# B&R Automation Studio project Project
Automation Studio 4.10

## Configuration BufferedFub

CPU PC_any, AutomationRuntime B4.92, Build 6.3.0, Vc V4.72.5

### Task classes (Cpu.sw)
```
Cyclic#1 (cycle 10000 us, tolerance 0 us):
  BufferFub_ <- BufferedFub.BufferFub_c-api_c-api.BufferFub_0.prg
  BufferF2_ <- BufferedFub.BufferFub2_c-api_c-api.BufferFub2_0.prg
Binaries: FWRules, udbdef, TCData, target, arconfig, User, sysconf, Role, iomap, asfw, ashwac, ashwd, components
Libraries: BufferFub, ExData, runtime, FileIO, AsIoTime, sys_lib, astime, exos, asieccon, exdeploy, astcp, BufferFub2
```

### Hardware
```
PC : PC_any v1.1.1.0 (OrderNumber=PC)
  ConfigurationID = Project_BufferedFub
  Cyclic1Duration = 10000
  Cyclic1Tolerance = 0
  Cyclic2Duration = 20000
  Cyclic2Tolerance = 0
  FileDevice1
  FileDeviceName1 = USER
  FileDevicePath1 = USER_PATH
  ActivateOpcUa = 1
  OpcUaPort = 4841
  OpcUaInformationModels_PV_Version = 1
```

### components.exoscomponent - PC/exosTechnology/components.exoscomponent
```
Element gBufferFub_0 (Type=exoscomponent)
  PackageSelection = Logical\BufferedFub\BufferFub_c-api_c-api\BufferFub.exospkg
  ErrorHandling = Component
  RestartEvent = Component
  StartupTimeout = 0
  Predefined:
    Files:
      File[0]:
        FileName = Linux\exos-comp-bufferfub_1.0.0_amd64.deb
        ChangeEvent = Reinstall
    Services:
      Service[0]:
        Type = Runtime
        Command = ./bufferfub
        WorkingDirectory = /home/user/bufferfub
      Service[1]:
        Type = Install
        Command = dpkg -i exos-comp-bufferfub_1.0.0_amd64.deb
        WorkingDirectory
      Service[2]:
        Type = Remove
        Command = dpkg --purge exos-comp-bufferfub
        WorkingDirectory
Element gBufferFub2_0 (Type=exoscomponent)
  PackageSelection = Logical\BufferedFub\BufferFub2_c-api_c-api\BufferFub2.exospkg
  ErrorHandling = Component
  RestartEvent = Component
  StartupTimeout = 0
  Predefined:
    Files:
      File[0]:
        FileName = Linux\exos-comp-bufferfub2_1.0.0_amd64.deb
        ChangeEvent = Reinstall
    Services:
      Service[0]:
        Type = Runtime
        Command = ./bufferfub2
        WorkingDirectory = /home/user/bufferfub2
      Service[1]:
        Type = Install
        Command = dpkg -i exos-comp-bufferfub2_1.0.0_amd64.deb
        WorkingDirectory
      Service[2]:
        Type = Remove
        Command = dpkg --purge exos-comp-bufferfub2
        WorkingDirectory
```

### target.exostarget - PC/exosTechnology/target.exostarget
```
Element gTarget_0 (Type=exostarget)
  General:
    ConnectionIP = 192.168.137.2
    Logging:
      LogLevel = Debug
      LogFilters:
        LogFilterUser = On
        LogFilterSystem = On
        LogFilterVerbose = On
      LogDestination = Volatile
    Deployment = On
      MaxRestarts = 10
    DataConnection = On
      ConnectionType = SharedMemory
      TimeSynchronization:
        TimeConnection:
          TimePort = 49001
        PrecisionUsec = 100
        GuardTimeSec = 4
        DeviationPerHourUsec = 100000
      DataConnectionLogging:
        LogConnection:
          LogPort = 49002
          LogShmPath = exos_log
        LogCycleTimeMsec = 100
  Components:
    ComponentsGeneral:
      ComponentsHeartbeatMsec = 500
      ComponentsTimeoutSec = 2
      ComponentsTaskClass = 2
      ComponentsCycleTimeMsec = 100
    Component[0]:
      ComponentConfigurationLink = gBufferFub_0
      DataModels:
        Instance[0]:
          InstanceName = BufferFub_0
          InstanceConnection:
            InstancePort = 49003
            InstanceShmPath = BufferFub_0
    Component[1]:
      ComponentConfigurationLink = gBufferFub2_0
      DataModels:
        Instance[0]:
          InstanceName = BufferFub2_0
          InstanceConnection:
            InstancePort = 49004
            InstanceShmPath = BufferFub2_0
  ComponentDataConnection:
    Version = 2.1.0-1
    ErrorHandling = Target
    RestartEvent = Target
    StartupTimeout = 5
    Predefined:
      Files:
        File[0]:
          FileName = ufw-exos-data
          ChangeEvent = Ignore
        File[1]:
          FileName = exos-data-ufw-profile.sh
          ChangeEvent = Ignore
        File[2]:
          FileName = exos-data-ports-allow.sh
          ChangeEvent = Restart
        File[3]:
          FileName = exos-data.conf
          ChangeEvent = Restart
        File[4]:
          FileName = exos-data_2.1.0-1_amd64.deb
          ChangeEvent = Reinstall
        File[5]:
          FileName = exos-data-eth_2.1.0-1_amd64.deb
          ChangeEvent = Reinstall
        File[6]:
          FileName = exos-data-remove.sh
          ChangeEvent = Ignore
        File[7]:
          FileName = run_server.sh
          ChangeEvent = Ignore
        File[8]:
          FileName = setup_build_environment.sh
          ChangeEvent = Ignore
        File[9]:
          FileName = libzmq5_4.2.1-4+deb9u2_amd64.deb
          ChangeEvent = Reinstall
        File[10]:
          FileName = libpgm-5.2-0_5.2.122~dfsg-2_amd64.deb
          ChangeEvent = Reinstall
        File[11]:
          FileName = libsodium18_1.0.11-2_amd64.deb
          ChangeEvent = Reinstall
      Services:
        Service[0]:
          Type = Install
          Command = dpkg -i *.deb
          WorkingDirectory
        Service[1]:
          Type = Remove
          Command = dpkg --purge exos-data
          WorkingDirectory
        Service[2]:
          Type = Remove
          Command = dpkg --purge exos-data-eth
          WorkingDirectory
        Service[3]:
          Type = Remove
          Command = sh exos-data-remove.sh
          WorkingDirectory
        Service[4]:
          Type = Startup
          Command = cp exos-data.conf /etc/exos-data.conf
          WorkingDirectory
        Service[5]:
          Type = Startup
          Command = sh exos-data-ufw-profile.sh
          WorkingDirectory
        Service[6]:
          Type = Startup
          Command = sh exos-data-ports-allow.sh
          WorkingDirectory
        Service[7]:
          Type = Runtime
          Command = /usr/bin/exos_mr
          WorkingDirectory
  Simulation:
    SimConnectionIP = 127.0.0.1
    SimDeployment = On
    SimDataConnection = On
      SimConnectionType = TCPIP
      SimTimeSynchronization:
        SimPrecisionUsec = 1000000
        SimGuardTimeSec = 30
    SimComponentsGeneral:
      SimComponentsHeartbeatMsec = 1000
      SimComponentsTimeoutSec = 75
```

## Logical view

- BufferFub.exospkg - exOS package description (not shown)

### Program Logical/BufferedFub/BufferFub_c-api_c-api/BufferFub_0 (IEC) - BufferFub application

#### BufferFub.var - BufferFub variable declaration
```iecst
VAR
    BufferFubInit_0 : BufferFubInit;
    BufferFubCyclic_0 : BufferFubCyclic;
    BufferFubExit_0 : BufferFubExit;
    BufferFubBufferUpdate_0 : BufferFubBufferUpdate;
    BufferFub_0 : BufferFub;
    ExComponentInfo_0 : ExComponentInfo;
    ExDatamodelInfo_0 : ExDatamodelInfo;
END_VAR
```

#### BufferFub.st - BufferFub application
```iecst
PROGRAM _INIT

    BufferFubInit_0();

END_PROGRAM

PROGRAM _CYCLIC

    //Auto connect:
    //BufferFubCyclic_0.Enable := ExComponentInfo_0.Operational; // Component has been deployed and started up successfully

    BufferFubCyclic_0(Handle := BufferFubInit_0.Handle, pBufferFub := ADR(BufferFub_0));

    BufferFubBufferUpdate_0.BufferHandle := BufferFubInit_0.bufferedSampleBufferHandle;
    UpdateBufferSampleSingle;
    //UpdateBufferSampleAll;

    ExComponentInfo_0(ExTargetLink := ADR(gTarget_0), ExComponentLink := ADR(gBufferFub_0), Enable := TRUE);

    ExDatamodelInfo_0(ExTargetLink := ADR(gTarget_0), Enable := TRUE, InstanceName := 'BufferFub_0');

END_PROGRAM

PROGRAM _EXIT

    BufferFubExit_0(Handle := BufferFubInit_0.Handle);

END_PROGRAM
```

#### UpdateBufferActions.st - BufferFub buffer actions
```iecst
(*Read a single change on BufferFubBufferUpdate_0.BufferHandle per scan*)
ACTION UpdateBufferSampleSingle:
    BufferFubBufferUpdate_0(UpdateDataset := TRUE);

    IF BufferFubBufferUpdate_0.DatasetUpdated THEN

        (* Your code here *)

    END_IF
END_ACTION

(*Read all changes on BufferFubBufferUpdate_0.BufferHandle within a single scan*)
ACTION UpdateBufferSampleAll:

    BufferFubBufferUpdate_0(UpdateDataset := FALSE); // update PendingUpdates without requesting UpdateDataset

    WHILE BufferFubBufferUpdate_0.PendingUpdates > 0 DO

        BufferFubBufferUpdate_0(UpdateDataset := TRUE);

        (* Your code here *)

    END_WHILE
END_ACTION
```

### Library Logical/BufferedFub/BufferFub_c-api_c-api/BufferFub (ANSIC) - BufferFub exOS library
Depends on: ExData

#### BufferFub.fun - BufferFub function blocks
```iecst
FUNCTION_BLOCK BufferFubInit
	VAR_OUTPUT
		Handle : UDINT;
		bufferedSampleBufferHandle : UDINT; (*Initialized BufferHandle for bufferedSample. Bufferhandle is linked to data in Cyclic*)
	END_VAR
	VAR
		_state : USINT;
	END_VAR
END_FUNCTION_BLOCK

FUNCTION_BLOCK BufferFubCyclic
	VAR_INPUT
		Enable : BOOL;
		Handle : UDINT;
		Start : BOOL;
		pBufferFub : REFERENCE TO BufferFub;
	END_VAR
	VAR_OUTPUT
		Active : BOOL;
		Error : BOOL;
		Disconnected : BOOL;
		Connected : BOOL;
		Operational : BOOL;
		Aborted : BOOL;
	END_VAR
	VAR
		_state : USINT;
	END_VAR
END_FUNCTION_BLOCK

FUNCTION_BLOCK BufferFubExit
	VAR_INPUT
		Handle : UDINT;
	END_VAR
	VAR
		_state : USINT;
	END_VAR
END_FUNCTION_BLOCK

FUNCTION_BLOCK BufferFubBufferUpdate (*Must be called in same TC as Cyclic. This function block finalizes in one scan and can be used for several different buffers*)
	VAR_INPUT
		BufferHandle : UDINT; (*Set this to the correct bufferhandle (from Init function block) before calling action UpdateBufferSampleSingle or UpdateBufferSampleAll*)
		UpdateDataset : BOOL; (*Set to TRUE to update dataset, PendingUpdates and OverflowErrors. Set to FALSE to only update PendingUpdates and OverflowErrors for BufferHandle without updating dataset*)
	END_VAR
	VAR_OUTPUT
		Error : BOOL; (*Set in case BufferHandle is invalid*)
		DatasetUpdated : BOOL; (*Set if dataset was updated successfully. Only when UpdateDataset is set to TRUE and there is something in the buffer*)
		PendingUpdates : UDINT; (*Number of datasets waiting in the buffer*)
		OverflowErrors : UDINT; (*Number of overflow errors which occurs when the buffer is full and new data arrives from GPOS*)
	END_VAR
END_FUNCTION_BLOCK
```

#### bufferfub.c - BufferFub library source
```c
#include <BufferFub.h>

#define EXOS_ASSERT_LOG &handle->logger
#define EXOS_ASSERT_CALLBACK inst->_state = 255;
#include "exos_log.h"
#include "exos_bufferfub.h"
#include <string.h>

#define SUCCESS(_format_, ...) exos_log_success(&handle->logger, EXOS_LOG_TYPE_USER, _format_, ##__VA_ARGS__);
#define INFO(_format_, ...) exos_log_info(&handle->logger, EXOS_LOG_TYPE_USER, _format_, ##__VA_ARGS__);
#define VERBOSE(_format_, ...) exos_log_debug(&handle->logger, EXOS_LOG_TYPE_USER + EXOS_LOG_TYPE_VERBOSE, _format_, ##__VA_ARGS__);
#define ERROR(_format_, ...) exos_log_error(&handle->logger, _format_, ##__VA_ARGS__);

typedef struct
{
    void *self;
    void* pData;
    size_t dataSize;
    void* databuffer;
    size_t bufferSize;
    size_t head;
    size_t tail;
    size_t overflowErrors;
} BufferFubBufferHandle_t;

typedef struct
{
    void *self;
    exos_log_handle_t logger;
    BufferFub data;

    exos_datamodel_handle_t bufferfub;

    exos_dataset_handle_t bufferedsample;
    BufferFubBufferHandle_t bufferedsample_buffer;
    exos_dataset_handle_t setup_dataset;
    exos_dataset_handle_t cmdsendburst;
} BufferFubHandle_t;

static int BufferFubBufferPush(BufferFubBufferHandle_t* bufferHandle, void* data)
{
    if (NULL == bufferHandle)
    {
        return -1;
    }
    if ((void *)bufferHandle != bufferHandle->self)
    {
        return -1;
    }
    if (((bufferHandle->head + 1) % bufferHandle->bufferSize) == bufferHandle->tail)
    {
        return -1;
    }

    memcpy(bufferHandle->databuffer + (bufferHandle->head * bufferHandle->dataSize), data, bufferHandle->dataSize);
    bufferHandle->head = (bufferHandle->head + 1) % bufferHandle->bufferSize;

    return 0;
}

static void datasetEvent(exos_dataset_handle_t *dataset, EXOS_DATASET_EVENT_TYPE event_type, void *info)
{
    struct BufferFubCyclic *inst = (struct BufferFubCyclic *)dataset->datamodel->user_context;
    BufferFubHandle_t *handle = (BufferFubHandle_t *)inst->Handle;

    switch (event_type)
    {
    case EXOS_DATASET_EVENT_UPDATED:
        VERBOSE("dataset %s updated! latency (us):%i", dataset->name, (exos_datamodel_get_nettime(dataset->datamodel) - dataset->nettime));
        //handle each subscription dataset separately
        if(0 == strcmp(dataset->name, "bufferedSample"))
        {
            //inst->pBufferFub->bufferedSample = *(UDINT *)dataset->data;

            if(BufferFubBufferPush(&handle->bufferedsample_buffer, dataset->data))
            {
                handle->bufferedsample_buffer.overflowErrors++;
                ERROR("Buffer overflow in bufferedSample update");
            }
        }
        break;

    case EXOS_DATASET_EVENT_PUBLISHED:
        VERBOSE("dataset %s published to local server for distribution! send buffer free:%i", dataset->name, dataset->send_buffer.free);
        //handle each published dataset separately
        if(0 == strcmp(dataset->name, "setup"))
        {
            // BufferFubSetup_typ *setup_dataset = (BufferFubSetup_typ *)dataset->data;
        }
        else if(0 == strcmp(dataset->name, "cmdSendBurst"))
        {
            // BOOL *cmdsendburst = (BOOL *)dataset->data;
        }
        break;

    case EXOS_DATASET_EVENT_DELIVERED:
        VERBOSE("dataset %s delivered to remote server for distribution! send buffer free:%i", dataset->name, dataset->send_buffer.free);
        //handle each published dataset separately
        if(0 == strcmp(dataset->name, "setup"))
        {
            // BufferFubSetup_typ *setup_dataset = (BufferFubSetup_typ *)dataset->data;
        }
        else if(0 == strcmp(dataset->name, "cmdSendBurst"))
        {
            // BOOL *cmdsendburst = (BOOL *)dataset->data;
        }
        break;

    case EXOS_DATASET_EVENT_CONNECTION_CHANGED:
        INFO("dataset %s changed state to %s", dataset->name, exos_get_state_string(dataset->connection_state));

        switch (dataset->connection_state)
        {
        case EXOS_STATE_DISCONNECTED:
            break;
        case EXOS_STATE_CONNECTED:
            //call the dataset changed event to update the dataset when connected
            //datasetEvent(dataset,EXOS_DATASET_UPDATED,info);
            break;
        case EXOS_STATE_OPERATIONAL:
            break;
        case EXOS_STATE_ABORTED:
            ERROR("dataset %s error %d (%s) occured", dataset->name, dataset->error, exos_get_error_string(dataset->error));
            break;
        }
        break;
    }

}

static void datamodelEvent(exos_datamodel_handle_t *datamodel, const EXOS_DATAMODEL_EVENT_TYPE event_type, void *info)
{
    struct BufferFubCyclic *inst = (struct BufferFubCyclic *)datamodel->user_context;
    BufferFubHandle_t *handle = (BufferFubHandle_t *)inst->Handle;

    switch (event_type)
    {
    case EXOS_DATAMODEL_EVENT_CONNECTION_CHANGED:
        INFO("application changed state to %s", exos_get_state_string(datamodel->connection_state));

        inst->Disconnected = 0;
        inst->Connected = 0;
        inst->Operational = 0;
        inst->Aborted = 0;

        switch (datamodel->connection_state)
        {
        case EXOS_STATE_DISCONNECTED:
            inst->Disconnected = 1;
            inst->_state = 255;
            break;
        case EXOS_STATE_CONNECTED:
            inst->Connected = 1;
            break;
        case EXOS_STATE_OPERATIONAL:
            SUCCESS("BufferFub operational!");
            inst->Operational = 1;
            break;
        case EXOS_STATE_ABORTED:
            ERROR("application error %d (%s) occured", datamodel->error, exos_get_error_string(datamodel->error));
            inst->_state = 255;
            inst->Aborted = 1;
            break;
        }
        break;
    case EXOS_DATAMODEL_EVENT_SYNC_STATE_CHANGED:
        break;

    default:
        break;

    }

}

_BUR_PUBLIC void BufferFubInit(struct BufferFubInit *inst)
{
    BufferFubHandle_t *handle;
    TMP_alloc(sizeof(BufferFubHandle_t), (void **)&handle);
    if (NULL == handle)
    {
        inst->Handle = 0;
        return;
    }

    memset(&handle->data, 0, sizeof(handle->data));
    handle->self = handle;

    // buffered alloc
    handle->bufferedsample_buffer.pData = 0; // set in BufferFubCyclic
    handle->bufferedsample_buffer.dataSize = sizeof(handle->data.bufferedSample);
    handle->bufferedsample_buffer.bufferSize = 20; // Note that empty is head==tail, thus only bufferSize-1 entries may be used.
    TMP_alloc(handle->bufferedsample_buffer.dataSize * handle->bufferedsample_buffer.bufferSize, (void **)&handle->bufferedsample_buffer.databuffer);
    if (NULL == handle->bufferedsample_buffer.databuffer)
    {
        inst->bufferedSampleBufferHandle = 0;
        TMP_free(sizeof(BufferFubHandle_t), (void *)handle);
        inst->Handle = 0;
        return;
    }

    handle->bufferedsample_buffer.head = 0;
    handle->bufferedsample_buffer.tail = 0;
    handle->bufferedsample_buffer.overflowErrors = 0;
    memset(handle->bufferedsample_buffer.databuffer, 0, handle->bufferedsample_buffer.dataSize * handle->bufferedsample_buffer.bufferSize);
    inst->bufferedSampleBufferHandle = &handle->bufferedsample_buffer;
    handle->bufferedsample_buffer.self = &handle->bufferedsample_buffer;

    exos_log_init(&handle->logger, "gBufferFub_0");

    exos_datamodel_handle_t *bufferfub = &handle->bufferfub;
    exos_dataset_handle_t *bufferedsample = &handle->bufferedsample;
    exos_dataset_handle_t *setup_dataset = &handle->setup_dataset;
    exos_dataset_handle_t *cmdsendburst = &handle->cmdsendburst;
    EXOS_ASSERT_OK(exos_datamodel_init(bufferfub, "BufferFub_0", "gBufferFub_0"));

    EXOS_ASSERT_OK(exos_dataset_init(bufferedsample, bufferfub, "bufferedSample", &handle->data.bufferedSample, sizeof(handle->data.bufferedSample)));
    EXOS_ASSERT_OK(exos_dataset_init(setup_dataset, bufferfub, "setup", &handle->data.setup, sizeof(handle->data.setup)));
    EXOS_ASSERT_OK(exos_dataset_init(cmdsendburst, bufferfub, "cmdSendBurst", &handle->data.cmdSendBurst, sizeof(handle->data.cmdSendBurst)));

    inst->Handle = (UDINT)handle;
}

_BUR_PUBLIC void BufferFubBufferUpdate(struct BufferFubBufferUpdate* inst)
{
    inst->DatasetUpdated = false;
    inst->Error = false;
    inst->OverflowErrors = 0;
    inst->PendingUpdates = 0;

    BufferFubBufferHandle_t *bufferHandle =  (BufferFubBufferHandle_t *)inst->BufferHandle;
    if (NULL == bufferHandle)
    {
        inst->Error = true;
        return;
    }
    if ((void *)bufferHandle != bufferHandle->self)
    {
        inst->Error = true;
        return;
    }

    inst->Error = false;
    inst->OverflowErrors = bufferHandle->overflowErrors;

    if(inst->UpdateDataset)
    {
        if (bufferHandle->tail == bufferHandle->head) // empty
        {
            inst->DatasetUpdated = false;
        }
        else
        {
            if(NULL != bufferHandle->pData)
            {
                memcpy(bufferHandle->pData, bufferHandle->databuffer + (bufferHandle->tail * bufferHandle->dataSize), bufferHandle->dataSize);
                //void* handle = bufferHandle->data[bufferHandle->tail];
                //should we set 0? bufferHandle->data[bufferHandle->tail] = NULL;
                bufferHandle->tail = (bufferHandle->tail + 1) % bufferHandle->bufferSize;
                inst->DatasetUpdated = true;
            }
            else
            {
                inst->Error = true;
                inst->DatasetUpdated = false;
            }
        }
    }
    else
    {
        inst->DatasetUpdated = false;
    }

    if (bufferHandle->tail > bufferHandle->head)
        inst->PendingUpdates = bufferHandle->bufferSize - (bufferHandle->tail - bufferHandle->head);
    else
        inst->PendingUpdates = bufferHandle->head - bufferHandle->tail;
}

_BUR_PUBLIC void BufferFubCyclic(struct BufferFubCyclic *inst)
{
    BufferFubHandle_t *handle = (BufferFubHandle_t *)inst->Handle;

    inst->Error = false;
    if (NULL == handle || NULL == inst->pBufferFub)
    {
        inst->Error = true;
        return;
    }
    if ((void *)handle != handle->self)
    {
        inst->Error = true;
        return;
    }

    // setup buffer address for xUpdate FUB:
    handle->bufferedsample_buffer.pData = &inst->pBufferFub->bufferedSample;

    BufferFub *data = &handle->data;
    exos_datamodel_handle_t *bufferfub = &handle->bufferfub;
    //the user context of the datamodel points to the BufferFubCyclic instance
    bufferfub->user_context = inst; //set it cyclically in case the program using the FUB is retransferred
    bufferfub->user_tag = 0; //user defined
    //handle online download of the library
    if(NULL != bufferfub->datamodel_event_callback && bufferfub->datamodel_event_callback != datamodelEvent)
    {
        bufferfub->datamodel_event_callback = datamodelEvent;
        exos_log_delete(&handle->logger);
        exos_log_init(&handle->logger, "gBufferFub_0");
    }

    exos_dataset_handle_t *bufferedsample = &handle->bufferedsample;
    bufferedsample->user_context = NULL; //user defined
    bufferedsample->user_tag = 0; //user defined
    //handle online download of the library
    if(NULL != bufferedsample->dataset_event_callback && bufferedsample->dataset_event_callback != datasetEvent)
    {
        bufferedsample->dataset_event_callback = datasetEvent;
    }

    exos_dataset_handle_t *setup_dataset = &handle->setup_dataset;
    setup_dataset->user_context = NULL; //user defined
    setup_dataset->user_tag = 0; //user defined
    //handle online download of the library
    if(NULL != setup_dataset->dataset_event_callback && setup_dataset->dataset_event_callback != datasetEvent)
    {
        setup_dataset->dataset_event_callback = datasetEvent;
    }

    exos_dataset_handle_t *cmdsendburst = &handle->cmdsendburst;
    cmdsendburst->user_context = NULL; //user defined
    cmdsendburst->user_tag = 0; //user defined
    //handle online download of the library
    if(NULL != cmdsendburst->dataset_event_callback && cmdsendburst->dataset_event_callback != datasetEvent)
    {
        cmdsendburst->dataset_event_callback = datasetEvent;
    }

    //unregister on disable
    if (inst->_state && !inst->Enable)
    {
        inst->_state = 255;
    }

    switch (inst->_state)
    {
    case 0:
        inst->Disconnected = 1;
        inst->Connected = 0;
        inst->Operational = 0;
        inst->Aborted = 0;

        if (inst->Enable)
        {
            inst->_state = 10;
        }
        break;

    case 10:
        inst->_state = 100;

        SUCCESS("starting BufferFub application..");

        //connect the datamodel, then the datasets
        EXOS_ASSERT_OK(exos_datamodel_connect_bufferfub(bufferfub, datamodelEvent));
        EXOS_ASSERT_OK(exos_dataset_connect(bufferedsample, EXOS_DATASET_SUBSCRIBE, datasetEvent));
        EXOS_ASSERT_OK(exos_dataset_connect(setup_dataset, EXOS_DATASET_PUBLISH, datasetEvent));
        EXOS_ASSERT_OK(exos_dataset_connect(cmdsendburst, EXOS_DATASET_PUBLISH, datasetEvent));

        inst->Active = true;
        break;

    case 100:
    case 101:
        if (inst->Start)
        {
            if (inst->_state == 100)
            {
                EXOS_ASSERT_OK(exos_datamodel_set_operational(bufferfub));
                inst->_state = 101;
            }
        }
        else
        {
            inst->_state = 100;
        }

        EXOS_ASSERT_OK(exos_datamodel_process(bufferfub));
        //put your cyclic code here!

        //publish the setup_dataset dataset as soon as there are changes
        if (0 != memcmp(&inst->pBufferFub->setup, &data->setup, sizeof(data->setup)))
        {
            memcpy(&data->setup, &inst->pBufferFub->setup, sizeof(data->setup));
            exos_dataset_publish(setup_dataset);
        }
        //publish the cmdsendburst dataset as soon as there are changes
        if (inst->pBufferFub->cmdSendBurst != data->cmdSendBurst)
        {
            data->cmdSendBurst = inst->pBufferFub->cmdSendBurst;
            exos_dataset_publish(cmdsendburst);
        }

        break;

    case 255:
        //disconnect the datamodel
        EXOS_ASSERT_OK(exos_datamodel_disconnect(bufferfub));

        inst->Active = false;
        inst->_state = 254;
        //no break

    case 254:
        if (!inst->Enable)
            inst->_state = 0;
        break;
    }

    exos_log_process(&handle->logger);

}

_BUR_PUBLIC void BufferFubExit(struct BufferFubExit *inst)
{
    BufferFubHandle_t *handle = (BufferFubHandle_t *)inst->Handle;

    if (NULL == handle)
    {
        ERROR("BufferFubExit: NULL handle, cannot delete resources");
        return;
    }
    if ((void *)handle != handle->self)
    {
        ERROR("BufferFubExit: invalid handle, cannot delete resources");
        return;
    }

    exos_datamodel_handle_t *bufferfub = &handle->bufferfub;

    EXOS_ASSERT_OK(exos_datamodel_delete(bufferfub));

    //delete buffer:
    BufferFubBufferHandle_t *bufferHandle =  (BufferFubBufferHandle_t *)&handle->bufferedsample_buffer;
    if (NULL == bufferHandle)
    {
        ERROR("BufferFubExit: NULL bufferhandle, cannot delete resources");
        return;
    }
    if ((void *)bufferHandle != bufferHandle->self)
    {
        ERROR("BufferFubExit: invalid bufferhandle, cannot delete resources");
        return;
    }

    //finish with deleting the log
    exos_log_delete(&handle->logger);
    //free the allocated handle
    TMP_free(sizeof(BufferFubHandle_t), (void *)handle);
}
```

### Package Logical/BufferedFub/BufferFub_c-api_c-api/Linux - BufferFub Linux resources

### bufferfub.c
```c
#include <unistd.h>
#include <string.h>
#include "termination.h"

#define EXOS_ASSERT_LOG &logger
#include "exos_log.h"
#include "exos_bufferfub.h"

#define SUCCESS(_format_, ...) exos_log_success(&logger, EXOS_LOG_TYPE_USER, _format_, ##__VA_ARGS__);
#define INFO(_format_, ...) exos_log_info(&logger, EXOS_LOG_TYPE_USER, _format_, ##__VA_ARGS__);
#define VERBOSE(_format_, ...) exos_log_debug(&logger, EXOS_LOG_TYPE_USER + EXOS_LOG_TYPE_VERBOSE, _format_, ##__VA_ARGS__);
#define ERROR(_format_, ...) exos_log_error(&logger, _format_, ##__VA_ARGS__);

exos_log_handle_t logger;

typedef struct {
    BufferFub *data;

    exos_datamodel_handle_t* bufferfub;

    exos_dataset_handle_t* bufferedsample;
    exos_dataset_handle_t* setup_dataset;
    exos_dataset_handle_t* cmdsendburst;
} application_info_t;

static void datasetEvent(exos_dataset_handle_t *dataset, EXOS_DATASET_EVENT_TYPE event_type, void *info)
{
    switch (event_type)
    {
    case EXOS_DATASET_EVENT_UPDATED:
        VERBOSE("dataset %s updated! latency (us):%i", dataset->name, (exos_datamodel_get_nettime(dataset->datamodel) - dataset->nettime));
        //handle each subscription dataset separately
        if(0 == strcmp(dataset->name,"setup"))
        {
            BufferFubSetup_typ *setup_dataset = (BufferFubSetup_typ *)dataset->data;
        }
        else if(0 == strcmp(dataset->name,"cmdSendBurst"))
        {
            bool *cmdsendburst = (bool *)dataset->data;

            if (*cmdsendburst){

                application_info_t *application = (application_info_t *)dataset->user_context;
                if (NULL != application)
                {
                    VERBOSE("Send burst, sampleCount=%u, sampleDelay=%u  ", application->data->setup.sampleCount, application->data->setup.sampleDelay);

                    for (size_t i = 0; i < application->data->setup.sampleCount; i++)
                    {
                        application->data->bufferedSample = i + 1;
                        exos_dataset_publish(application->bufferedsample);

                        usleep(application->data->setup.sampleDelay);
                    }
                }
            }
        }
        break;

    case EXOS_DATASET_EVENT_PUBLISHED:
        VERBOSE("dataset %s published to local server for distribution! send buffer free:%i", dataset->name, dataset->send_buffer.free);
        //handle each published dataset separately
        if(0 == strcmp(dataset->name, "bufferedSample"))
        {
            uint32_t *bufferedsample = (uint32_t *)dataset->data;
        }
        break;

    case EXOS_DATASET_EVENT_DELIVERED:
        VERBOSE("dataset %s delivered to remote server for distribution! send buffer free:%i", dataset->name, dataset->send_buffer.free);
        //handle each published dataset separately
        if(0 == strcmp(dataset->name, "bufferedSample"))
        {
            uint32_t *bufferedsample = (uint32_t *)dataset->data;
        }
        break;

    case EXOS_DATASET_EVENT_CONNECTION_CHANGED:
        INFO("dataset %s changed state to %s", dataset->name, exos_get_state_string(dataset->connection_state));

        switch (dataset->connection_state)
        {
        case EXOS_STATE_DISCONNECTED:
            break;
        case EXOS_STATE_CONNECTED:
            //call the dataset changed event to update the dataset when connected
            //datasetEvent(dataset,EXOS_DATASET_UPDATED,info);
            break;
        case EXOS_STATE_OPERATIONAL:
            break;
        case EXOS_STATE_ABORTED:
            ERROR("dataset %s error %d (%s) occured", dataset->name, dataset->error, exos_get_error_string(dataset->error));
            break;
        }
        break;
    }

}

static void datamodelEvent(exos_datamodel_handle_t *datamodel, const EXOS_DATAMODEL_EVENT_TYPE event_type, void *info)
{
    switch (event_type)
    {
    case EXOS_DATAMODEL_EVENT_CONNECTION_CHANGED:
        INFO("application changed state to %s", exos_get_state_string(datamodel->connection_state));

        switch (datamodel->connection_state)
        {
        case EXOS_STATE_DISCONNECTED:
            break;
        case EXOS_STATE_CONNECTED:
            break;
        case EXOS_STATE_OPERATIONAL:
            SUCCESS("BufferFub operational!");
            break;
        case EXOS_STATE_ABORTED:
            ERROR("application error %d (%s) occured", datamodel->error, exos_get_error_string(datamodel->error));
            break;
        }
        break;
    case EXOS_DATAMODEL_EVENT_SYNC_STATE_CHANGED:
        break;

    default:
        break;

    }

}

int main()
{
    BufferFub data;

    exos_datamodel_handle_t bufferfub;

    exos_dataset_handle_t bufferedsample;
    exos_dataset_handle_t setup_dataset;
    exos_dataset_handle_t cmdsendburst;

    application_info_t myapplication = {&data, &bufferfub, &bufferedsample, &setup_dataset, &cmdsendburst};

    exos_log_init(&logger, "gBufferFub_0");

    SUCCESS("starting BufferFub application..");

    EXOS_ASSERT_OK(exos_datamodel_init(&bufferfub, "BufferFub_0", "gBufferFub_0"));

    //set the user_context to access custom data in the callbacks
    bufferfub.user_context = NULL; //user defined
    bufferfub.user_tag = 0; //user defined

    EXOS_ASSERT_OK(exos_dataset_init(&bufferedsample, &bufferfub, "bufferedSample", &data.bufferedSample, sizeof(data.bufferedSample)));
    bufferedsample.user_context = NULL; //user defined
    bufferedsample.user_tag = 0; //user defined

    EXOS_ASSERT_OK(exos_dataset_init(&setup_dataset, &bufferfub, "setup", &data.setup, sizeof(data.setup)));
    setup_dataset.user_context = NULL; //user defined
    setup_dataset.user_tag = 0; //user defined

    EXOS_ASSERT_OK(exos_dataset_init(&cmdsendburst, &bufferfub, "cmdSendBurst", &data.cmdSendBurst, sizeof(data.cmdSendBurst)));
    cmdsendburst.user_context = &myapplication; //user defined
    cmdsendburst.user_tag = 0; //user defined

    //connect the datamodel
    EXOS_ASSERT_OK(exos_datamodel_connect_bufferfub(&bufferfub, datamodelEvent));

    //connect datasets
    EXOS_ASSERT_OK(exos_dataset_connect(&bufferedsample, EXOS_DATASET_PUBLISH, datasetEvent));
    EXOS_ASSERT_OK(exos_dataset_connect(&setup_dataset, EXOS_DATASET_SUBSCRIBE, datasetEvent));
    EXOS_ASSERT_OK(exos_dataset_connect(&cmdsendburst, EXOS_DATASET_SUBSCRIBE, datasetEvent));

    catch_termination();
    while (true)
    {
        EXOS_ASSERT_OK(exos_datamodel_process(&bufferfub));
        exos_log_process(&logger);

        //put your cyclic code here!

        if (is_terminated())
        {
            SUCCESS("BufferFub application terminated, closing..");
            break;
        }
    }

    EXOS_ASSERT_OK(exos_datamodel_delete(&bufferfub));

    //finish with deleting the log
    exos_log_delete(&logger);
    return 0;
}
```

- BufferFub2.exospkg - exOS package description (not shown)

### Program Logical/BufferedFub/BufferFub2_c-api_c-api/BufferFub2_0 (IEC) - BufferFub2 application

#### BufferFub2.var - BufferFub2 variable declaration
```iecst
VAR
    BufferFub2Init_0 : BufferFub2Init;
    BufferFub2Cyclic_0 : BufferFub2Cyclic;
    BufferFub2Exit_0 : BufferFub2Exit;
    BufferFub2BufferUpdate_0 : BufferFub2BufferUpdate;
    BufferFub2_0 : BufferFub2;
    ExComponentInfo_0 : ExComponentInfo;
    ExDatamodelInfo_0 : ExDatamodelInfo;
END_VAR
```

#### BufferFub2.st - BufferFub2 application
```iecst
PROGRAM _INIT

    BufferFub2Init_0();

END_PROGRAM

PROGRAM _CYCLIC

    //Auto connect:
    //BufferFub2Cyclic_0.Enable := ExComponentInfo_0.Operational; // Component has been deployed and started up successfully

    BufferFub2Cyclic_0(Handle := BufferFub2Init_0.Handle, pBufferFub2 := ADR(BufferFub2_0));

    BufferFub2BufferUpdate_0.BufferHandle := BufferFub2Init_0.bufferedSampleBufferHandle;
    UpdateBufferSampleSingle;
    //UpdateBufferSampleAll;

    ExComponentInfo_0(ExTargetLink := ADR(gTarget_0), ExComponentLink := ADR(gBufferFub2_0), Enable := TRUE);

    ExDatamodelInfo_0(ExTargetLink := ADR(gTarget_0), Enable := TRUE, InstanceName := 'BufferFub2_0');

END_PROGRAM

PROGRAM _EXIT

    BufferFub2Exit_0(Handle := BufferFub2Init_0.Handle);

END_PROGRAM
```

#### UpdateBufferActions.st - BufferFub2 buffer actions
```iecst
(*Read a single change on BufferFub2BufferUpdate_0.BufferHandle per scan*)
ACTION UpdateBufferSampleSingle:
    BufferFub2BufferUpdate_0(UpdateDataset := TRUE);

    IF BufferFub2BufferUpdate_0.DatasetUpdated THEN

        (* Your code here *)

    END_IF
END_ACTION

(*Read all changes on BufferFub2BufferUpdate_0.BufferHandle within a single scan*)
ACTION UpdateBufferSampleAll:

    BufferFub2BufferUpdate_0(UpdateDataset := FALSE); // update PendingUpdates without requesting UpdateDataset

    WHILE BufferFub2BufferUpdate_0.PendingUpdates > 0 DO

        BufferFub2BufferUpdate_0(UpdateDataset := TRUE);

        (* Your code here *)

    END_WHILE
END_ACTION
```

### Library Logical/BufferedFub/BufferFub2_c-api_c-api/BufferFub2 (ANSIC) - BufferFub2 exOS library
Depends on: ExData

#### BufferFub2.typ - BufferFub2 datamodel declaration
```iecst
TYPE
	BufferFub2Setup_typ : 	STRUCT
		sampleCount : UDINT; (*number of samples sent each time cmdSendBurst is set*)
		sampleDelay : UDINT; (*ms between samples*)
	END_STRUCT;
	BufferFub2SubStruct_typ : 	STRUCT
		moreid : UDINT; (*id number*)
		moredata : REAL; (*some data*)
	END_STRUCT;
	BufferFub2Sample_typ : 	STRUCT
		id : UDINT; (*id number*)
		data : REAL; (*some data*)
		subStruct : BufferFub2SubStruct_typ; (*a sub structure*)
	END_STRUCT;
	BufferFub2 : 	STRUCT
		bufferedSample : BufferFub2Sample_typ; (*SUB BUFFERED*)
		setup : BufferFub2Setup_typ; (*PUB*)
		cmdSendBurst : BOOL; (*PUB*)
	END_STRUCT;
END_TYPE
```

#### BufferFub2.fun - BufferFub2 function blocks
```iecst
FUNCTION_BLOCK BufferFub2Init
	VAR_OUTPUT
		Handle : UDINT;
		bufferedSampleBufferHandle : UDINT; (*Initialized BufferHandle for bufferedSample. Bufferhandle is linked to data in Cyclic*)
	END_VAR
	VAR
		_state : USINT;
	END_VAR
END_FUNCTION_BLOCK

FUNCTION_BLOCK BufferFub2Cyclic
	VAR_INPUT
		Enable : BOOL;
		Handle : UDINT;
		Start : BOOL;
		pBufferFub2 : REFERENCE TO BufferFub2;
	END_VAR
	VAR_OUTPUT
		Active : BOOL;
		Error : BOOL;
		Disconnected : BOOL;
		Connected : BOOL;
		Operational : BOOL;
		Aborted : BOOL;
	END_VAR
	VAR
		_state : USINT;
	END_VAR
END_FUNCTION_BLOCK

FUNCTION_BLOCK BufferFub2Exit
	VAR_INPUT
		Handle : UDINT;
	END_VAR
	VAR
		_state : USINT;
	END_VAR
END_FUNCTION_BLOCK

FUNCTION_BLOCK BufferFub2BufferUpdate (*Must be called in same TC as Cyclic. This function block finalizes in one scan and can be used for several different buffers*)
	VAR_INPUT
		BufferHandle : UDINT; (*Set this to the correct bufferhandle (from Init function block) before calling action UpdateBufferSampleSingle or UpdateBufferSampleAll*)
		UpdateDataset : BOOL; (*Set to TRUE to update dataset, PendingUpdates and OverflowErrors. Set to FALSE to only update PendingUpdates and OverflowErrors for BufferHandle without updating dataset*)
	END_VAR
	VAR_OUTPUT
		Error : BOOL; (*Set in case BufferHandle is invalid*)
		DatasetUpdated : BOOL; (*Set if dataset was updated successfully. Only when UpdateDataset is set to TRUE and there is something in the buffer*)
		PendingUpdates : UDINT; (*Number of datasets waiting in the buffer*)
		OverflowErrors : UDINT; (*Number of overflow errors which occurs when the buffer is full and new data arrives from GPOS*)
	END_VAR
END_FUNCTION_BLOCK
```

#### bufferfub2.c - BufferFub2 library source
```c
#include <BufferFub2.h>

#define EXOS_ASSERT_LOG &handle->logger
#define EXOS_ASSERT_CALLBACK inst->_state = 255;
#include "exos_log.h"
#include "exos_bufferfub2.h"
#include <string.h>

#define SUCCESS(_format_, ...) exos_log_success(&handle->logger, EXOS_LOG_TYPE_USER, _format_, ##__VA_ARGS__);
#define INFO(_format_, ...) exos_log_info(&handle->logger, EXOS_LOG_TYPE_USER, _format_, ##__VA_ARGS__);
#define VERBOSE(_format_, ...) exos_log_debug(&handle->logger, EXOS_LOG_TYPE_USER + EXOS_LOG_TYPE_VERBOSE, _format_, ##__VA_ARGS__);
#define ERROR(_format_, ...) exos_log_error(&handle->logger, _format_, ##__VA_ARGS__);

typedef struct
{
    void *self;
    void* pData;
    size_t dataSize;
    void* databuffer;
    size_t bufferSize;
    size_t head;
    size_t tail;
    size_t overflowErrors;
} BufferFub2BufferHandle_t;

typedef struct
{
    void *self;
    exos_log_handle_t logger;
    BufferFub2 data;

    exos_datamodel_handle_t bufferfub2;

    exos_dataset_handle_t bufferedsample;
    BufferFub2BufferHandle_t bufferedsample_buffer;
    exos_dataset_handle_t setup_dataset;
    exos_dataset_handle_t cmdsendburst;
} BufferFub2Handle_t;

static int BufferFub2BufferPush(BufferFub2BufferHandle_t* bufferHandle, void* data)
{
    if (NULL == bufferHandle)
    {
        return -1;
    }
    if ((void *)bufferHandle != bufferHandle->self)
    {
        return -1;
    }
    if (((bufferHandle->head + 1) % bufferHandle->bufferSize) == bufferHandle->tail)
    {
        return -1;
    }

    memcpy(bufferHandle->databuffer + (bufferHandle->head * bufferHandle->dataSize), data, bufferHandle->dataSize);
    bufferHandle->head = (bufferHandle->head + 1) % bufferHandle->bufferSize;

    return 0;
}

static void datasetEvent(exos_dataset_handle_t *dataset, EXOS_DATASET_EVENT_TYPE event_type, void *info)
{
    struct BufferFub2Cyclic *inst = (struct BufferFub2Cyclic *)dataset->datamodel->user_context;
    BufferFub2Handle_t *handle = (BufferFub2Handle_t *)inst->Handle;

    switch (event_type)
    {
    case EXOS_DATASET_EVENT_UPDATED:
        VERBOSE("dataset %s updated! latency (us):%i", dataset->name, (exos_datamodel_get_nettime(dataset->datamodel) - dataset->nettime));
        //handle each subscription dataset separately
        if(0 == strcmp(dataset->name, "bufferedSample"))
        {
            if(BufferFub2BufferPush(&handle->bufferedsample_buffer, dataset->data))
            {
                handle->bufferedsample_buffer.overflowErrors++;
                ERROR("Buffer overflow in bufferedSample update");
            }
        }
        break;

    case EXOS_DATASET_EVENT_PUBLISHED:
        VERBOSE("dataset %s published to local server for distribution! send buffer free:%i", dataset->name, dataset->send_buffer.free);
        //handle each published dataset separately
        if(0 == strcmp(dataset->name, "setup"))
        {
            // BufferFub2Setup_typ *setup_dataset = (BufferFub2Setup_typ *)dataset->data;
        }
        else if(0 == strcmp(dataset->name, "cmdSendBurst"))
        {
            // BOOL *cmdsendburst = (BOOL *)dataset->data;
        }
        break;

    case EXOS_DATASET_EVENT_DELIVERED:
        VERBOSE("dataset %s delivered to remote server for distribution! send buffer free:%i", dataset->name, dataset->send_buffer.free);
        //handle each published dataset separately
        if(0 == strcmp(dataset->name, "setup"))
        {
            // BufferFub2Setup_typ *setup_dataset = (BufferFub2Setup_typ *)dataset->data;
        }
        else if(0 == strcmp(dataset->name, "cmdSendBurst"))
        {
            // BOOL *cmdsendburst = (BOOL *)dataset->data;
        }
        break;

    case EXOS_DATASET_EVENT_CONNECTION_CHANGED:
        INFO("dataset %s changed state to %s", dataset->name, exos_get_state_string(dataset->connection_state));

        switch (dataset->connection_state)
        {
        case EXOS_STATE_DISCONNECTED:
            break;
        case EXOS_STATE_CONNECTED:
            //call the dataset changed event to update the dataset when connected
            //datasetEvent(dataset,EXOS_DATASET_UPDATED,info);
            break;
        case EXOS_STATE_OPERATIONAL:
            break;
        case EXOS_STATE_ABORTED:
            ERROR("dataset %s error %d (%s) occured", dataset->name, dataset->error, exos_get_error_string(dataset->error));
            break;
        }
        break;
    }

}

static void datamodelEvent(exos_datamodel_handle_t *datamodel, const EXOS_DATAMODEL_EVENT_TYPE event_type, void *info)
{
    struct BufferFub2Cyclic *inst = (struct BufferFub2Cyclic *)datamodel->user_context;
    BufferFub2Handle_t *handle = (BufferFub2Handle_t *)inst->Handle;

    switch (event_type)
    {
    case EXOS_DATAMODEL_EVENT_CONNECTION_CHANGED:
        INFO("application changed state to %s", exos_get_state_string(datamodel->connection_state));

        inst->Disconnected = 0;
        inst->Connected = 0;
        inst->Operational = 0;
        inst->Aborted = 0;

        switch (datamodel->connection_state)
        {
        case EXOS_STATE_DISCONNECTED:
            inst->Disconnected = 1;
            inst->_state = 255;
            break;
        case EXOS_STATE_CONNECTED:
            inst->Connected = 1;
            break;
        case EXOS_STATE_OPERATIONAL:
            SUCCESS("BufferFub2 operational!");
            inst->Operational = 1;
            break;
        case EXOS_STATE_ABORTED:
            ERROR("application error %d (%s) occured", datamodel->error, exos_get_error_string(datamodel->error));
            inst->_state = 255;
            inst->Aborted = 1;
            break;
        }
        break;
    case EXOS_DATAMODEL_EVENT_SYNC_STATE_CHANGED:
        break;

    default:
        break;

    }

}

_BUR_PUBLIC void BufferFub2Init(struct BufferFub2Init *inst)
{
    BufferFub2Handle_t *handle;
    TMP_alloc(sizeof(BufferFub2Handle_t), (void **)&handle);
    if (NULL == handle)
    {
        inst->Handle = 0;
        return;
    }

    memset(&handle->data, 0, sizeof(handle->data));
    handle->self = handle;

    // Allocation and initialization of buffer(s)
    handle->bufferedsample_buffer.pData = 0; // set in BufferFub2Cyclic
    handle->bufferedsample_buffer.dataSize = sizeof(handle->data.bufferedSample);
    handle->bufferedsample_buffer.bufferSize = 20; // Note that empty is head==tail, thus only bufferSize-1 entries may be used.
    TMP_alloc(handle->bufferedsample_buffer.dataSize * handle->bufferedsample_buffer.bufferSize, (void **)&handle->bufferedsample_buffer.databuffer);
    if (NULL == handle->bufferedsample_buffer.databuffer)
    {
        inst->bufferedSampleBufferHandle = 0;
        TMP_free(sizeof(BufferFub2Handle_t), (void *)handle);
        inst->Handle = 0;
        return;
    }

    handle->bufferedsample_buffer.head = 0;
    handle->bufferedsample_buffer.tail = 0;
    handle->bufferedsample_buffer.overflowErrors = 0;
    memset(handle->bufferedsample_buffer.databuffer, 0, handle->bufferedsample_buffer.dataSize * handle->bufferedsample_buffer.bufferSize);
    inst->bufferedSampleBufferHandle = (UDINT)&handle->bufferedsample_buffer;
    handle->bufferedsample_buffer.self = &handle->bufferedsample_buffer;

    exos_log_init(&handle->logger, "gBufferFub2_0");

    exos_datamodel_handle_t *bufferfub2 = &handle->bufferfub2;
    exos_dataset_handle_t *bufferedsample = &handle->bufferedsample;
    exos_dataset_handle_t *setup_dataset = &handle->setup_dataset;
    exos_dataset_handle_t *cmdsendburst = &handle->cmdsendburst;
    EXOS_ASSERT_OK(exos_datamodel_init(bufferfub2, "BufferFub2_0", "gBufferFub2_0"));

    EXOS_ASSERT_OK(exos_dataset_init(bufferedsample, bufferfub2, "bufferedSample", &handle->data.bufferedSample, sizeof(handle->data.bufferedSample)));
    EXOS_ASSERT_OK(exos_dataset_init(setup_dataset, bufferfub2, "setup", &handle->data.setup, sizeof(handle->data.setup)));
    EXOS_ASSERT_OK(exos_dataset_init(cmdsendburst, bufferfub2, "cmdSendBurst", &handle->data.cmdSendBurst, sizeof(handle->data.cmdSendBurst)));

    inst->Handle = (UDINT)handle;
}

_BUR_PUBLIC void BufferFub2BufferUpdate(struct BufferFub2BufferUpdate* inst)
{
    inst->DatasetUpdated = false;
    inst->Error = false;
    inst->OverflowErrors = 0;
    inst->PendingUpdates = 0;

    BufferFub2BufferHandle_t *bufferHandle =  (BufferFub2BufferHandle_t *)inst->BufferHandle;
    if (NULL == bufferHandle)
    {
        inst->Error = true;
        return;
    }
    if ((void *)bufferHandle != bufferHandle->self)
    {
        inst->Error = true;
        return;
    }

    inst->Error = false;
    inst->OverflowErrors = bufferHandle->overflowErrors;

    if(inst->UpdateDataset)
    {
        if (bufferHandle->tail == bufferHandle->head) // empty
        {
            inst->DatasetUpdated = false;
        }
        else
        {
            if(NULL != bufferHandle->pData)
            {
                memcpy(bufferHandle->pData, bufferHandle->databuffer + (bufferHandle->tail * bufferHandle->dataSize), bufferHandle->dataSize);
                //void* handle = bufferHandle->data[bufferHandle->tail];
                //should we set 0? bufferHandle->data[bufferHandle->tail] = NULL;
                bufferHandle->tail = (bufferHandle->tail + 1) % bufferHandle->bufferSize;
                inst->DatasetUpdated = true;
            }
            else
            {
                inst->Error = true;
                inst->DatasetUpdated = false;
            }
        }
    }
    else
    {
        inst->DatasetUpdated = false;
    }

    if (bufferHandle->tail > bufferHandle->head)
        inst->PendingUpdates = bufferHandle->bufferSize - (bufferHandle->tail - bufferHandle->head);
    else
        inst->PendingUpdates = bufferHandle->head - bufferHandle->tail;
}

_BUR_PUBLIC void BufferFub2Cyclic(struct BufferFub2Cyclic *inst)
{
    BufferFub2Handle_t *handle = (BufferFub2Handle_t *)inst->Handle;

    inst->Error = false;
    if (NULL == handle || NULL == inst->pBufferFub2)
    {
        inst->Error = true;
        return;
    }
    if ((void *)handle != handle->self)
    {
        inst->Error = true;
        return;
    }

    // setup buffer address(es) for BufferFub2Update:
    handle->bufferedsample_buffer.pData = &inst->pBufferFub2->bufferedSample;

    BufferFub2 *data = &handle->data;
    exos_datamodel_handle_t *bufferfub2 = &handle->bufferfub2;
    //the user context of the datamodel points to the BufferFub2Cyclic instance
    bufferfub2->user_context = inst; //set it cyclically in case the program using the FUB is retransferred
    bufferfub2->user_tag = 0; //user defined
    //handle online download of the library
    if(NULL != bufferfub2->datamodel_event_callback && bufferfub2->datamodel_event_callback != datamodelEvent)
    {
        bufferfub2->datamodel_event_callback = datamodelEvent;
        exos_log_delete(&handle->logger);
        exos_log_init(&handle->logger, "gBufferFub2_0");
    }

    exos_dataset_handle_t *bufferedsample = &handle->bufferedsample;
    bufferedsample->user_context = NULL; //user defined
    bufferedsample->user_tag = 0; //user defined
    //handle online download of the library
    if(NULL != bufferedsample->dataset_event_callback && bufferedsample->dataset_event_callback != datasetEvent)
    {
        bufferedsample->dataset_event_callback = datasetEvent;
    }

    exos_dataset_handle_t *setup_dataset = &handle->setup_dataset;
    setup_dataset->user_context = NULL; //user defined
    setup_dataset->user_tag = 0; //user defined
    //handle online download of the library
    if(NULL != setup_dataset->dataset_event_callback && setup_dataset->dataset_event_callback != datasetEvent)
    {
        setup_dataset->dataset_event_callback = datasetEvent;
    }

    exos_dataset_handle_t *cmdsendburst = &handle->cmdsendburst;
    cmdsendburst->user_context = NULL; //user defined
    cmdsendburst->user_tag = 0; //user defined
    //handle online download of the library
    if(NULL != cmdsendburst->dataset_event_callback && cmdsendburst->dataset_event_callback != datasetEvent)
    {
        cmdsendburst->dataset_event_callback = datasetEvent;
    }

    //unregister on disable
    if (inst->_state && !inst->Enable)
    {
        inst->_state = 255;
    }

    switch (inst->_state)
    {
    case 0:
        inst->Disconnected = 1;
        inst->Connected = 0;
        inst->Operational = 0;
        inst->Aborted = 0;

        if (inst->Enable)
        {
            inst->_state = 10;
        }
        break;

    case 10:
        inst->_state = 100;

        SUCCESS("starting BufferFub2 application..");

        //connect the datamodel, then the datasets
        EXOS_ASSERT_OK(exos_datamodel_connect_bufferfub2(bufferfub2, datamodelEvent));
        EXOS_ASSERT_OK(exos_dataset_connect(bufferedsample, EXOS_DATASET_SUBSCRIBE, datasetEvent));
        EXOS_ASSERT_OK(exos_dataset_connect(setup_dataset, EXOS_DATASET_PUBLISH, datasetEvent));
        EXOS_ASSERT_OK(exos_dataset_connect(cmdsendburst, EXOS_DATASET_PUBLISH, datasetEvent));

        inst->Active = true;
        break;

    case 100:
    case 101:
        if (inst->Start)
        {
            if (inst->_state == 100)
            {
                EXOS_ASSERT_OK(exos_datamodel_set_operational(bufferfub2));
                inst->_state = 101;
            }
        }
        else
        {
            inst->_state = 100;
        }

        EXOS_ASSERT_OK(exos_datamodel_process(bufferfub2));
        //put your cyclic code here!

        //publish the setup_dataset dataset as soon as there are changes
        if (0 != memcmp(&inst->pBufferFub2->setup, &data->setup, sizeof(data->setup)))
        {
            memcpy(&data->setup, &inst->pBufferFub2->setup, sizeof(data->setup));
            exos_dataset_publish(setup_dataset);
        }
        //publish the cmdsendburst dataset as soon as there are changes
        if (inst->pBufferFub2->cmdSendBurst != data->cmdSendBurst)
        {
            data->cmdSendBurst = inst->pBufferFub2->cmdSendBurst;
            exos_dataset_publish(cmdsendburst);
        }

        break;

    case 255:
        //disconnect the datamodel
        EXOS_ASSERT_OK(exos_datamodel_disconnect(bufferfub2));

        inst->Active = false;
        inst->_state = 254;
        //no break

    case 254:
        if (!inst->Enable)
            inst->_state = 0;
        break;
    }

    exos_log_process(&handle->logger);

}

_BUR_PUBLIC void BufferFub2Exit(struct BufferFub2Exit *inst)
{
    BufferFub2Handle_t *handle = (BufferFub2Handle_t *)inst->Handle;

    if (NULL == handle)
    {
        ERROR("BufferFub2Exit: NULL handle, cannot delete resources");
        return;
    }
    if ((void *)handle != handle->self)
    {
        ERROR("BufferFub2Exit: invalid handle, cannot delete resources");
        return;
    }

    exos_datamodel_handle_t *bufferfub2 = &handle->bufferfub2;

    EXOS_ASSERT_OK(exos_datamodel_delete(bufferfub2));

    //delete buffer(s):
    BufferFub2BufferHandle_t *bufferHandle =  (BufferFub2BufferHandle_t *)&handle->bufferedsample_buffer;
    if (NULL == bufferHandle)
    {
        ERROR("BufferFub2Exit: NULL bufferhandle, cannot delete resources");
        return;
    }
    if ((void *)bufferHandle != bufferHandle->self)
    {
        ERROR("BufferFub2Exit: invalid bufferhandle, cannot delete resources");
        return;
    }

    //finish with deleting the log
    exos_log_delete(&handle->logger);
    //free the allocated handle
    TMP_free(sizeof(BufferFub2Handle_t), (void *)handle);
}
```

### Package Logical/BufferedFub/BufferFub2_c-api_c-api/Linux - BufferFub2 Linux resources

### exos_bufferfub2.h - Generated datamodel header for BufferFub2
```c
/*Automatically generated header file from BufferFub2.typ*/

#ifndef _EXOS_COMP_BUFFERFUB2_H_
#define _EXOS_COMP_BUFFERFUB2_H_

#include "exos_api.h"

#if defined(_SG4)
#include <BufferFub2.h>
#else
#include <stddef.h>
#include <stdint.h>
#include <stdbool.h>

typedef struct BufferFub2Setup_typ
{
    uint32_t sampleCount; //number of samples sent each time cmdSendBurst is set
    uint32_t sampleDelay; //ms between samples

} BufferFub2Setup_typ;

typedef struct BufferFub2SubStruct_typ
{
    uint32_t moreid; //id number
    float moredata; //some data

} BufferFub2SubStruct_typ;

typedef struct BufferFub2Sample_typ
{
    uint32_t id; //id number
    float data; //some data
    struct BufferFub2SubStruct_typ subStruct; //a sub structure

} BufferFub2Sample_typ;

typedef struct BufferFub2
{
    struct BufferFub2Sample_typ bufferedSample; //SUB BUFFERED
    struct BufferFub2Setup_typ setup; //PUB
    bool cmdSendBurst; //PUB

} BufferFub2;

#endif // _SG4

EXOS_ERROR_CODE exos_datamodel_connect_bufferfub2(exos_datamodel_handle_t *datamodel, exos_datamodel_event_cb datamodel_event_callback);

#endif // _EXOS_COMP_BUFFERFUB2_H_
```

### exos_bufferfub2.c - Generated datamodel source for BufferFub2
```c
/*Automatically generated c file from BufferFub2.typ*/

#include "exos_bufferfub2.h"

const char config_bufferfub2[] = "{\"name\":\"struct\",\"attributes\":{\"name\":\"<NAME>\",\"dataType\":\"BufferFub2\",\"info\":\"<infoId0>\"},\"children\":[{\"name\":\"struct\",\"attributes\":{\"name\":\"bufferedSample\",\"dataType\":\"BufferFub2Sample_typ\",\"comment\":\"SUB\",\"info\":\"<infoId1>\"},\"children\":[{\"name\":\"variable\",\"attributes\":{\"name\":\"id\",\"dataType\":\"UDINT\",\"info\":\"<infoId2>\"}},{\"name\":\"variable\",\"attributes\":{\"name\":\"data\",\"dataType\":\"REAL\",\"info\":\"<infoId3>\"}},{\"name\":\"struct\",\"attributes\":{\"name\":\"subStruct\",\"dataType\":\"BufferFub2SubStruct_typ\",\"info\":\"<infoId4>\"},\"children\":[{\"name\":\"variable\",\"attributes\":{\"name\":\"moreid\",\"dataType\":\"UDINT\",\"info\":\"<infoId5>\"}},{\"name\":\"variable\",\"attributes\":{\"name\":\"moredata\",\"dataType\":\"REAL\",\"info\":\"<infoId6>\"}}]}]},{\"name\":\"struct\",\"attributes\":{\"name\":\"setup\",\"dataType\":\"BufferFub2Setup_typ\",\"comment\":\"PUB\",\"info\":\"<infoId7>\"},\"children\":[{\"name\":\"variable\",\"attributes\":{\"name\":\"sampleCount\",\"dataType\":\"UDINT\",\"info\":\"<infoId8>\"}},{\"name\":\"variable\",\"attributes\":{\"name\":\"sampleDelay\",\"dataType\":\"UDINT\",\"info\":\"<infoId9>\"}}]},{\"name\":\"variable\",\"attributes\":{\"name\":\"cmdSendBurst\",\"dataType\":\"BOOL\",\"comment\":\"PUB\",\"info\":\"<infoId10>\"}}]}";

/*Connect the BufferFub2 datamodel to the server*/
EXOS_ERROR_CODE exos_datamodel_connect_bufferfub2(exos_datamodel_handle_t *datamodel, exos_datamodel_event_cb datamodel_event_callback)
{
    BufferFub2 data;
    exos_dataset_info_t datasets[] = {
        {EXOS_DATASET_BROWSE_NAME_INIT,{}},
        {EXOS_DATASET_BROWSE_NAME(bufferedSample),{}},
        {EXOS_DATASET_BROWSE_NAME(bufferedSample.id),{}},
        {EXOS_DATASET_BROWSE_NAME(bufferedSample.data),{}},
        {EXOS_DATASET_BROWSE_NAME(bufferedSample.subStruct),{}},
        {EXOS_DATASET_BROWSE_NAME(bufferedSample.subStruct.moreid),{}},
        {EXOS_DATASET_BROWSE_NAME(bufferedSample.subStruct.moredata),{}},
        {EXOS_DATASET_BROWSE_NAME(setup),{}},
        {EXOS_DATASET_BROWSE_NAME(setup.sampleCount),{}},
        {EXOS_DATASET_BROWSE_NAME(setup.sampleDelay),{}},
        {EXOS_DATASET_BROWSE_NAME(cmdSendBurst),{}}
    };

    exos_datamodel_calc_dataset_info(datasets, sizeof(datasets));

    return exos_datamodel_connect(datamodel, config_bufferfub2, datasets, sizeof(datasets), datamodel_event_callback);
}
```

### bufferfub2.c - Linux application
```c
#include <unistd.h>
#include <string.h>
#include "termination.h"

#define EXOS_ASSERT_LOG &logger
#include "exos_log.h"
#include "exos_bufferfub2.h"

#define SUCCESS(_format_, ...) exos_log_success(&logger, EXOS_LOG_TYPE_USER, _format_, ##__VA_ARGS__);
#define INFO(_format_, ...) exos_log_info(&logger, EXOS_LOG_TYPE_USER, _format_, ##__VA_ARGS__);
#define VERBOSE(_format_, ...) exos_log_debug(&logger, EXOS_LOG_TYPE_USER + EXOS_LOG_TYPE_VERBOSE, _format_, ##__VA_ARGS__);
#define ERROR(_format_, ...) exos_log_error(&logger, _format_, ##__VA_ARGS__);

exos_log_handle_t logger;

static void datasetEvent(exos_dataset_handle_t *dataset, EXOS_DATASET_EVENT_TYPE event_type, void *info)
{
    switch (event_type)
    {
    case EXOS_DATASET_EVENT_UPDATED:
        VERBOSE("dataset %s updated! latency (us):%i", dataset->name, (exos_datamodel_get_nettime(dataset->datamodel) - dataset->nettime));
        //handle each subscription dataset separately
        if(0 == strcmp(dataset->name,"setup"))
        {
            BufferFub2Setup_typ *setup_dataset = (BufferFub2Setup_typ *)dataset->data;
        }
        else if(0 == strcmp(dataset->name,"cmdSendBurst"))
        {
            bool *cmdsendburst = (bool *)dataset->data;
        }
        break;

    case EXOS_DATASET_EVENT_PUBLISHED:
        VERBOSE("dataset %s published to local server for distribution! send buffer free:%i", dataset->name, dataset->send_buffer.free);
        //handle each published dataset separately
        if(0 == strcmp(dataset->name, "bufferedSample"))
        {
            BufferFub2Sample_typ *bufferedsample = (BufferFub2Sample_typ *)dataset->data;
        }
        break;

    case EXOS_DATASET_EVENT_DELIVERED:
        VERBOSE("dataset %s delivered to remote server for distribution! send buffer free:%i", dataset->name, dataset->send_buffer.free);
        //handle each published dataset separately
        if(0 == strcmp(dataset->name, "bufferedSample"))
        {
            BufferFub2Sample_typ *bufferedsample = (BufferFub2Sample_typ *)dataset->data;
        }
        break;

    case EXOS_DATASET_EVENT_CONNECTION_CHANGED:
        INFO("dataset %s changed state to %s", dataset->name, exos_get_state_string(dataset->connection_state));

        switch (dataset->connection_state)
        {
        case EXOS_STATE_DISCONNECTED:
            break;
        case EXOS_STATE_CONNECTED:
            //call the dataset changed event to update the dataset when connected
            //datasetEvent(dataset,EXOS_DATASET_UPDATED,info);
            break;
        case EXOS_STATE_OPERATIONAL:
            break;
        case EXOS_STATE_ABORTED:
            ERROR("dataset %s error %d (%s) occured", dataset->name, dataset->error, exos_get_error_string(dataset->error));
            break;
        }
        break;
    }

}

static void datamodelEvent(exos_datamodel_handle_t *datamodel, const EXOS_DATAMODEL_EVENT_TYPE event_type, void *info)
{
    switch (event_type)
    {
    case EXOS_DATAMODEL_EVENT_CONNECTION_CHANGED:
        INFO("application changed state to %s", exos_get_state_string(datamodel->connection_state));

        switch (datamodel->connection_state)
        {
        case EXOS_STATE_DISCONNECTED:
            break;
        case EXOS_STATE_CONNECTED:
            break;
        case EXOS_STATE_OPERATIONAL:
            SUCCESS("BufferFub2 operational!");
            break;
        case EXOS_STATE_ABORTED:
            ERROR("application error %d (%s) occured", datamodel->error, exos_get_error_string(datamodel->error));
            break;
        }
        break;
    case EXOS_DATAMODEL_EVENT_SYNC_STATE_CHANGED:
        break;

    default:
        break;

    }

}

int main()
{
    BufferFub2 data;

    exos_datamodel_handle_t bufferfub2;

    exos_dataset_handle_t bufferedsample;
    exos_dataset_handle_t setup_dataset;
    exos_dataset_handle_t cmdsendburst;

    exos_log_init(&logger, "gBufferFub2_0");

    SUCCESS("starting BufferFub2 application..");

    EXOS_ASSERT_OK(exos_datamodel_init(&bufferfub2, "BufferFub2_0", "gBufferFub2_0"));

    //set the user_context to access custom data in the callbacks
    bufferfub2.user_context = NULL; //user defined
    bufferfub2.user_tag = 0; //user defined

    EXOS_ASSERT_OK(exos_dataset_init(&bufferedsample, &bufferfub2, "bufferedSample", &data.bufferedSample, sizeof(data.bufferedSample)));
    bufferedsample.user_context = NULL; //user defined
    bufferedsample.user_tag = 0; //user defined

    EXOS_ASSERT_OK(exos_dataset_init(&setup_dataset, &bufferfub2, "setup", &data.setup, sizeof(data.setup)));
    setup_dataset.user_context = NULL; //user defined
    setup_dataset.user_tag = 0; //user defined

    EXOS_ASSERT_OK(exos_dataset_init(&cmdsendburst, &bufferfub2, "cmdSendBurst", &data.cmdSendBurst, sizeof(data.cmdSendBurst)));
    cmdsendburst.user_context = NULL; //user defined
    cmdsendburst.user_tag = 0; //user defined

    //connect the datamodel
    EXOS_ASSERT_OK(exos_datamodel_connect_bufferfub2(&bufferfub2, datamodelEvent));

    //connect datasets
    EXOS_ASSERT_OK(exos_dataset_connect(&bufferedsample, EXOS_DATASET_PUBLISH, datasetEvent));
    EXOS_ASSERT_OK(exos_dataset_connect(&setup_dataset, EXOS_DATASET_SUBSCRIBE, datasetEvent));
    EXOS_ASSERT_OK(exos_dataset_connect(&cmdsendburst, EXOS_DATASET_SUBSCRIBE, datasetEvent));

    catch_termination();
    while (true)
    {
        EXOS_ASSERT_OK(exos_datamodel_process(&bufferfub2));
        exos_log_process(&logger);

        //put your cyclic code here!

        if (is_terminated())
        {
            SUCCESS("BufferFub2 application terminated, closing..");
            break;
        }
    }

    EXOS_ASSERT_OK(exos_datamodel_delete(&bufferfub2));

    //finish with deleting the log
    exos_log_delete(&logger);
    return 0;
}
```

### CMakeLists.txt - CMake build file script
```
cmake_minimum_required(VERSION 3.0)

project(bufferfub2)

set(CMAKE_BUILD_TYPE Debug)
add_executable(bufferfub2 termination.c bufferfub2.c exos_bufferfub2.c)
target_include_directories(bufferfub2 PUBLIC ..)
target_link_libraries(bufferfub2 zmq exos-api)

install(TARGETS bufferfub2 RUNTIME DESTINATION /home/user/bufferfub2)

set(CPACK_GENERATOR "DEB")
set(CPACK_PACKAGE_NAME exos-comp-bufferfub2)
set(CPACK_PACKAGE_DESCRIPTION_SUMMARY "BufferFub2 summary")
set(CPACK_PACKAGE_DESCRIPTION "Some description")
set(CPACK_PACKAGE_VENDOR "Your Company")

set(CPACK_PACKAGE_VERSION_MAJOR 1)
set(CPACK_PACKAGE_VERSION_MINOR 0)
set(CPACK_PACKAGE_VERSION_PATCH 0)
set(CPACK_PACKAGE_FILE_NAME exos-comp-bufferfub2_1.0.0_amd64)
set(CPACK_DEBIAN_PACKAGE_MAINTAINER "Your Name")

set(CPACK_DEBIAN_PACKAGE_SHLIBDEPS ON)

include(CPack)
```

- build.sh - build file shell script (not shown)

- bufferfub2 - BufferFub2 application (binary file, 33072 bytes)
### Library Logical/BufferedFub/BufferFub_c-static_c-api/BufferFub (ANSIC)
Depends on: ExData

#### exos_bufferfub.h - Generated datamodel header for BufferFub
```c
/*Automatically generated header file from BufferFub.typ*/

#ifndef _EXOS_COMP_BUFFERFUB_H_
#define _EXOS_COMP_BUFFERFUB_H_

#include "exos_api.h"

#if defined(_SG4)
#include <BufferFub.h>
#else
#include <stddef.h>
#include <stdint.h>
#include <stdbool.h>

typedef struct BufferFubSetup_typ
{
    uint32_t sampleCount; //number of samples sent each time cmdSendBurst is set
    uint32_t sampleDelay; //ms between samples

} BufferFubSetup_typ;

typedef struct BufferFub
{
    uint32_t bufferedSample; //SUB BUFFERED
    struct BufferFubSetup_typ setup; //PUB
    bool cmdSendBurst; //PUB

} BufferFub;

#endif // _SG4

EXOS_ERROR_CODE exos_datamodel_connect_bufferfub(exos_datamodel_handle_t *datamodel, exos_datamodel_event_cb datamodel_event_callback);

#endif // _EXOS_COMP_BUFFERFUB_H_
```

#### libbufferfub.h - BufferFub static library wrapper header
```c
#ifndef _LIBBUFFERFUB_H_
#define _LIBBUFFERFUB_H_

#include "exos_bufferfub.h"

typedef void (*libBufferFub_event_cb)(void);
typedef void (*libBufferFub_method_fn)(void);
typedef int32_t (*libBufferFub_get_nettime_fn)(void);
typedef void (*libBufferFub_log_fn)(char *log_entry);

typedef struct libBufferFubbufferedSample
{
    libBufferFub_event_cb on_change;
    int32_t nettime;
    uint32_t value;
} libBufferFubbufferedSample_t;

typedef struct libBufferFubsetup
{
    libBufferFub_method_fn publish;
    BufferFubSetup_typ value;
} libBufferFubsetup_t;

typedef struct libBufferFubcmdSendBurst
{
    libBufferFub_method_fn publish;
    bool value;
} libBufferFubcmdSendBurst_t;

typedef struct libBufferFub_log
{
    libBufferFub_log_fn error;
    libBufferFub_log_fn warning;
    libBufferFub_log_fn success;
    libBufferFub_log_fn info;
    libBufferFub_log_fn debug;
    libBufferFub_log_fn verbose;
} libBufferFub_log_t;

typedef struct libBufferFub
{
    libBufferFub_method_fn connect;
    libBufferFub_method_fn disconnect;
    libBufferFub_method_fn process;
    libBufferFub_method_fn set_operational;
    libBufferFub_method_fn dispose;
    libBufferFub_get_nettime_fn get_nettime;
    libBufferFub_log_t log;
    libBufferFub_event_cb on_connected;
    libBufferFub_event_cb on_disconnected;
    libBufferFub_event_cb on_operational;
    bool is_connected;
    bool is_operational;
    libBufferFubbufferedSample_t bufferedSample;
    libBufferFubsetup_t setup;
    libBufferFubcmdSendBurst_t cmdSendBurst;
} libBufferFub_t;

#ifdef __cplusplus
extern "C" {
#endif
libBufferFub_t *libBufferFub_init(void);
#ifdef __cplusplus
}
#endif
#endif // _LIBBUFFERFUB_H_
```

### Program Logical/BufferedFub/BufferFub_c-static_c-api/BufferFub_0 (IEC)

#### BufferFub.var - BufferFub variable declaration
```iecst
VAR
    BufferFub_0 : BufferFub;
    BufferFubCyclic_0 : BufferFubCyclic;
    ExComponentInfo_0 : ExComponentInfo;
    ExDatamodelInfo_0 : ExDatamodelInfo;
END_VAR
```

### Program Logical/BufferedFub/BufferFub_c-static_c-api/Linux

#### bufferfub.c
```c
#include <unistd.h>
#include <string.h>
#include "termination.h"

#define EXOS_ASSERT_LOG &logger
#include "exos_log.h"
#include "exos_bufferfub.h"

#define SUCCESS(_format_, ...) exos_log_success(&logger, EXOS_LOG_TYPE_USER, _format_, ##__VA_ARGS__);
#define INFO(_format_, ...) exos_log_info(&logger, EXOS_LOG_TYPE_USER, _format_, ##__VA_ARGS__);
#define VERBOSE(_format_, ...) exos_log_debug(&logger, EXOS_LOG_TYPE_USER + EXOS_LOG_TYPE_VERBOSE, _format_, ##__VA_ARGS__);
#define ERROR(_format_, ...) exos_log_error(&logger, _format_, ##__VA_ARGS__);

exos_log_handle_t logger;

static void datasetEvent(exos_dataset_handle_t *dataset, EXOS_DATASET_EVENT_TYPE event_type, void *info)
{
    switch (event_type)
    {
    case EXOS_DATASET_EVENT_UPDATED:
        VERBOSE("dataset %s updated! latency (us):%i", dataset->name, (exos_datamodel_get_nettime(dataset->datamodel) - dataset->nettime));
        //handle each subscription dataset separately
        if(0 == strcmp(dataset->name,"setup"))
        {
            BufferFubSetup_typ *setup_dataset = (BufferFubSetup_typ *)dataset->data;
        }
        else if(0 == strcmp(dataset->name,"cmdSendBurst"))
        {
            bool *cmdsendburst = (bool *)dataset->data;
        }
        break;

    case EXOS_DATASET_EVENT_PUBLISHED:
        VERBOSE("dataset %s published to local server for distribution! send buffer free:%i", dataset->name, dataset->send_buffer.free);
        //handle each published dataset separately
        if(0 == strcmp(dataset->name, "bufferedSample"))
        {
            uint32_t *bufferedsample = (uint32_t *)dataset->data;
        }
        break;

    case EXOS_DATASET_EVENT_DELIVERED:
        VERBOSE("dataset %s delivered to remote server for distribution! send buffer free:%i", dataset->name, dataset->send_buffer.free);
        //handle each published dataset separately
        if(0 == strcmp(dataset->name, "bufferedSample"))
        {
            uint32_t *bufferedsample = (uint32_t *)dataset->data;
        }
        break;

    case EXOS_DATASET_EVENT_CONNECTION_CHANGED:
        INFO("dataset %s changed state to %s", dataset->name, exos_get_state_string(dataset->connection_state));

        switch (dataset->connection_state)
        {
        case EXOS_STATE_DISCONNECTED:
            break;
        case EXOS_STATE_CONNECTED:
            //call the dataset changed event to update the dataset when connected
            //datasetEvent(dataset,EXOS_DATASET_UPDATED,info);
            break;
        case EXOS_STATE_OPERATIONAL:
            break;
        case EXOS_STATE_ABORTED:
            ERROR("dataset %s error %d (%s) occured", dataset->name, dataset->error, exos_get_error_string(dataset->error));
            break;
        }
        break;
    }

}

static void datamodelEvent(exos_datamodel_handle_t *datamodel, const EXOS_DATAMODEL_EVENT_TYPE event_type, void *info)
{
    switch (event_type)
    {
    case EXOS_DATAMODEL_EVENT_CONNECTION_CHANGED:
        INFO("application changed state to %s", exos_get_state_string(datamodel->connection_state));

        switch (datamodel->connection_state)
        {
        case EXOS_STATE_DISCONNECTED:
            break;
        case EXOS_STATE_CONNECTED:
            break;
        case EXOS_STATE_OPERATIONAL:
            SUCCESS("BufferFub operational!");
            break;
        case EXOS_STATE_ABORTED:
            ERROR("application error %d (%s) occured", datamodel->error, exos_get_error_string(datamodel->error));
            break;
        }
        break;
    case EXOS_DATAMODEL_EVENT_SYNC_STATE_CHANGED:
        break;

    default:
        break;

    }

}

int main()
{
    BufferFub data;

    exos_datamodel_handle_t bufferfub;

    exos_dataset_handle_t bufferedsample;
    exos_dataset_handle_t setup_dataset;
    exos_dataset_handle_t cmdsendburst;

    exos_log_init(&logger, "gBufferFub_0");

    SUCCESS("starting BufferFub application..");

    EXOS_ASSERT_OK(exos_datamodel_init(&bufferfub, "BufferFub_0", "gBufferFub_0"));

    //set the user_context to access custom data in the callbacks
    bufferfub.user_context = NULL; //user defined
    bufferfub.user_tag = 0; //user defined

    EXOS_ASSERT_OK(exos_dataset_init(&bufferedsample, &bufferfub, "bufferedSample", &data.bufferedSample, sizeof(data.bufferedSample)));
    bufferedsample.user_context = NULL; //user defined
    bufferedsample.user_tag = 0; //user defined

    EXOS_ASSERT_OK(exos_dataset_init(&setup_dataset, &bufferfub, "setup", &data.setup, sizeof(data.setup)));
    setup_dataset.user_context = NULL; //user defined
    setup_dataset.user_tag = 0; //user defined

    EXOS_ASSERT_OK(exos_dataset_init(&cmdsendburst, &bufferfub, "cmdSendBurst", &data.cmdSendBurst, sizeof(data.cmdSendBurst)));
    cmdsendburst.user_context = NULL; //user defined
    cmdsendburst.user_tag = 0; //user defined

    //connect the datamodel
    EXOS_ASSERT_OK(exos_datamodel_connect_bufferfub(&bufferfub, datamodelEvent));

    //connect datasets
    EXOS_ASSERT_OK(exos_dataset_connect(&bufferedsample, EXOS_DATASET_PUBLISH, datasetEvent));
    EXOS_ASSERT_OK(exos_dataset_connect(&setup_dataset, EXOS_DATASET_SUBSCRIBE, datasetEvent));
    EXOS_ASSERT_OK(exos_dataset_connect(&cmdsendburst, EXOS_DATASET_SUBSCRIBE, datasetEvent));

    catch_termination();
    while (true)
    {
        EXOS_ASSERT_OK(exos_datamodel_process(&bufferfub));
        exos_log_process(&logger);

        //put your cyclic code here!

        if (is_terminated())
        {
            SUCCESS("BufferFub application terminated, closing..");
            break;
        }
    }

    EXOS_ASSERT_OK(exos_datamodel_delete(&bufferfub));

    //finish with deleting the log
    exos_log_delete(&logger);
    return 0;
}
```

#### CMakeLists.txt
```
cmake_minimum_required(VERSION 3.0)

project(bufferfub)

set(CMAKE_BUILD_TYPE Debug)
add_executable(bufferfub termination.c bufferfub.c exos_bufferfub.c)
target_include_directories(bufferfub PUBLIC ..)
target_link_libraries(bufferfub zmq exos-api)

install(TARGETS bufferfub RUNTIME DESTINATION /home/user/bufferfub)

set(CPACK_GENERATOR "DEB")
set(CPACK_PACKAGE_NAME exos-comp-bufferfub)
set(CPACK_PACKAGE_DESCRIPTION_SUMMARY "BufferFub summary")
set(CPACK_PACKAGE_DESCRIPTION "Some description")
set(CPACK_PACKAGE_VENDOR "Your Company")

set(CPACK_PACKAGE_VERSION_MAJOR 1)
set(CPACK_PACKAGE_VERSION_MINOR 0)
set(CPACK_PACKAGE_VERSION_PATCH 0)
set(CPACK_PACKAGE_FILE_NAME exos-comp-bufferfub_1.0.0_amd64)
set(CPACK_DEBIAN_PACKAGE_MAINTAINER "Your Name")

set(CPACK_DEBIAN_PACKAGE_SHLIBDEPS ON)

include(CPack)
```

### Library Logical/BufferedFub/BufferFub_cpp_c-api/BufferFub (ANSIC) - BufferFub exOS library
Depends on: ExData

#### exos_bufferfub.c - Generated datamodel source for BufferFub
```c
/*Automatically generated c file from BufferFub.typ*/

#include "exos_bufferfub.h"

const char config_bufferfub[] = "{\"name\":\"struct\",\"attributes\":{\"name\":\"<NAME>\",\"dataType\":\"BufferFub\",\"info\":\"<infoId0>\"},\"children\":[{\"name\":\"variable\",\"attributes\":{\"name\":\"bufferedSample\",\"dataType\":\"UDINT\",\"comment\":\"SUB\",\"info\":\"<infoId1>\"}},{\"name\":\"struct\",\"attributes\":{\"name\":\"setup\",\"dataType\":\"BufferFubSetup_typ\",\"comment\":\"PUB\",\"info\":\"<infoId2>\"},\"children\":[{\"name\":\"variable\",\"attributes\":{\"name\":\"sampleCount\",\"dataType\":\"UDINT\",\"info\":\"<infoId3>\"}},{\"name\":\"variable\",\"attributes\":{\"name\":\"sampleDelay\",\"dataType\":\"UDINT\",\"info\":\"<infoId4>\"}}]},{\"name\":\"variable\",\"attributes\":{\"name\":\"cmdSendBurst\",\"dataType\":\"BOOL\",\"comment\":\"PUB\",\"info\":\"<infoId5>\"}}]}";

/*Connect the BufferFub datamodel to the server*/
EXOS_ERROR_CODE exos_datamodel_connect_bufferfub(exos_datamodel_handle_t *datamodel, exos_datamodel_event_cb datamodel_event_callback)
{
    BufferFub data;
    exos_dataset_info_t datasets[] = {
        {EXOS_DATASET_BROWSE_NAME_INIT,{}},
        {EXOS_DATASET_BROWSE_NAME(bufferedSample),{}},
        {EXOS_DATASET_BROWSE_NAME(setup),{}},
        {EXOS_DATASET_BROWSE_NAME(setup.sampleCount),{}},
        {EXOS_DATASET_BROWSE_NAME(setup.sampleDelay),{}},
        {EXOS_DATASET_BROWSE_NAME(cmdSendBurst),{}}
    };

    exos_datamodel_calc_dataset_info(datasets, sizeof(datasets));

    return exos_datamodel_connect(datamodel, config_bufferfub, datasets, sizeof(datasets), datamodel_event_callback);
}
```

#### BufferFubDataset.hpp - BufferFub dataset class
```cpp
#if __GNUC__ == 4
#error ########## GCC 4.1.2 used but C++ Template Requires GCC 6.3 - Change the complier in the build options ##########
#endif
#ifndef _BUFFERFUBDATASET_H_
#define _BUFFERFUBDATASET_H_

#include <string>
#include <iostream>
#include <string.h>
#include <functional>

extern "C" {
    #include "exos_bufferfub.h"
}

#include "BufferFubLogger.hpp"
#define exos_assert_ok(_plog_,_exp_)                                                                                                    \
    do                                                                                                                                  \
    {                                                                                                                                   \
        EXOS_ERROR_CODE err = _exp_;                                                                                                    \
        if (EXOS_ERROR_OK != err)                                                                                                       \
        {                                                                                                                               \
            _plog_->error << "Error in file " << __FILE__ << ":" << __LINE__ << std::endl;                                               \
            _plog_->error << #_exp_ " returned " << err << " (" << exos_get_error_string(err) << ") instead of expected 0" << std::endl; \
        }                                                                                                                               \
    } while (0)

template <typename T>
class BufferFubDataset
{
private:
    exos_dataset_handle_t dataset = {};
    BufferFubLogger* log;
    std::function<void()> _onChange = [](){};
    void datasetEvent(exos_dataset_handle_t *dataset, EXOS_DATASET_EVENT_TYPE event_type, void *info) {
        switch (event_type)
        {
            case EXOS_DATASET_EVENT_UPDATED:
                log->verbose << "dataset " << dataset->name << " updated! latency (us):" << (exos_datamodel_get_nettime(dataset->datamodel) - dataset->nettime) << std::endl;
                nettime = dataset->nettime;
                _onChange();
                break;
            case EXOS_DATASET_EVENT_PUBLISHED:
                log->verbose << "dataset " << dataset->name << "  published to local server for distribution! send buffer free:" << dataset->send_buffer.free << std::endl;
                break;
            case EXOS_DATASET_EVENT_DELIVERED:
                log->verbose << "dataset " << dataset->name << " delivered to remote server for distribution! send buffer free:" << dataset->send_buffer.free << std::endl;
                break;
            case EXOS_DATASET_EVENT_CONNECTION_CHANGED:
                log->info << "dataset " << dataset->name << " changed state to " << exos_get_state_string(dataset->connection_state) << std::endl;

                switch (dataset->connection_state)
                {
                    case EXOS_STATE_DISCONNECTED:
                        break;
                    case EXOS_STATE_CONNECTED:
                        break;
                    case EXOS_STATE_OPERATIONAL:
                        break;
                    case EXOS_STATE_ABORTED:
                        log->error << "dataset " << dataset->name << " error " << dataset->error << " (" << exos_get_error_string(dataset->error) << ") occured" << std::endl;
                        break;
                }
                break;
        }
    }
    static void _datasetEvent(exos_dataset_handle_t *dataset, EXOS_DATASET_EVENT_TYPE event_type, void *info) {
        BufferFubDataset* inst = static_cast<BufferFubDataset*>(dataset->user_context);
        inst->datasetEvent(dataset, event_type, info);
    }

public:
    BufferFubDataset() {};

    T value;
    int nettime;
    void init(exos_datamodel_handle_t *datamodel, const char *browse_name, BufferFubLogger* _log) {
        log = _log;
        exos_assert_ok(log, exos_dataset_init(&dataset, datamodel, browse_name, &value, sizeof(value)));
        dataset.user_context = this;
    };
    void connect(EXOS_DATASET_TYPE type) {
        exos_assert_ok(log, exos_dataset_connect(&dataset, type, &BufferFubDataset::_datasetEvent));
    };
    void publish() {
        exos_dataset_publish(&dataset);
    };
    void onChange(std::function<void()> f) {_onChange = std::move(f);};

    ~BufferFubDataset() {
        exos_assert_ok(log, exos_dataset_delete(&dataset));
    };
};

#endif
```

#### BufferFubLogger.hpp - BufferFub logger class
```cpp
#ifndef _BUFFERFUB_LOGGER_H_
#define _BUFFERFUB_LOGGER_H_

#include <iostream>
#include <sstream>
#include <string>

extern "C" {
    #include "exos_log.h"
}

class ExosLogger
{
private:
    exos_log_handle_t* logger;
    EXOS_LOG_LEVEL logLevel;
    EXOS_LOG_TYPE logType;
    std::stringstream sstream;
public:
    typedef std::ostream&  (*ManipFn)(std::ostream&);
    typedef std::ios_base& (*FlagsFn)(std::ios_base&);

    ExosLogger(exos_log_handle_t* logger, EXOS_LOG_LEVEL logLevel, EXOS_LOG_TYPE logType);

    template<class T>  // int, double, strings, etc
        ExosLogger& operator<<(const T& output)
    {
        sstream << output;
        return *this;
    }

    ExosLogger& operator<<(ManipFn manip) /// endl, flush, setw, setfill, etc.
    {
        manip(sstream);

        if (manip == static_cast<ManipFn>(std::flush)
            || manip == static_cast<ManipFn>(std::endl ) )
            this->flush();

        return *this;
    }

    ExosLogger& operator<<(FlagsFn manip) /// setiosflags, resetiosflags
    {
        manip(sstream);
        return *this;
    }

    void flush();

    ExosLogger();
};

class BufferFubLogger
{
public:
    BufferFubLogger(std::string name)
        : info(&logger, EXOS_LOG_LEVEL_INFO, EXOS_LOG_TYPE_USER)
        , warning(&logger, EXOS_LOG_LEVEL_WARNING, EXOS_LOG_TYPE_USER)
        , error(&logger, EXOS_LOG_LEVEL_ERROR, EXOS_LOG_TYPE_USER)
        , debug(&logger, EXOS_LOG_LEVEL_DEBUG, EXOS_LOG_TYPE_USER)
        , verbose(&logger, EXOS_LOG_LEVEL_WARNING, EXOS_LOG_TYPE(EXOS_LOG_TYPE_USER+EXOS_LOG_TYPE_VERBOSE))
        , success(&logger, EXOS_LOG_LEVEL_SUCCESS, EXOS_LOG_TYPE_USER)
    {
        exos_log_init(&logger, name.c_str());
    };
    void process() {
        exos_log_process(&logger);
    }
    ~BufferFubLogger() {
        exos_log_delete(&logger);
    };
    ExosLogger info;
    ExosLogger warning;
    ExosLogger error;
    ExosLogger debug;
    ExosLogger verbose;
    ExosLogger success;
private:
    exos_log_handle_t logger = {};
};

#endif
```

#### BufferFubLogger.cpp - BufferFub logger class implementation
```cpp
#include "BufferFubLogger.hpp"

ExosLogger::ExosLogger(exos_log_handle_t* logger, EXOS_LOG_LEVEL logLevel, EXOS_LOG_TYPE logType)
    : logger(logger)
    , logLevel(logLevel)
    , logType(logType)
{
}

void ExosLogger::flush()
{
    switch(logLevel)
    {
        case EXOS_LOG_LEVEL_INFO:
            exos_log_info(logger, logType, const_cast<char*>(sstream.str().c_str()));
            break;
        case EXOS_LOG_LEVEL_DEBUG:
            exos_log_debug(logger, logType, const_cast<char*>(sstream.str().c_str()));
            break;
        case EXOS_LOG_LEVEL_ERROR:
            exos_log_error(logger, const_cast<char*>(sstream.str().c_str()));
            break;
        case EXOS_LOG_LEVEL_SUCCESS:
            exos_log_success(logger, logType, const_cast<char*>(sstream.str().c_str()));
            break;
        case EXOS_LOG_LEVEL_WARNING:
            exos_log_warning(logger, logType, const_cast<char*>(sstream.str().c_str()));
            break;
    }
    sstream.str(std::string());
    sstream.clear();
}
```


Listed in the project but not available here: Logical/Global.typ, Logical/Global.var, Logical/Libraries, Logical/Package, Logical/typfiles, Logical/BufferedFub/BufferFub_c-api_c-api/BufferFub/BufferFub.typ, Logical/BufferedFub/BufferFub_c-api_c-api/BufferFub/exos_bufferfub.h, Logical/BufferedFub/BufferFub_c-api_c-api/BufferFub/exos_bufferfub.c, Logical/BufferedFub/BufferFub_c-api_c-api/BufferFub/heapsize.cpp, Logical/BufferedFub/BufferFub2_c-api_c-api/BufferFub2/exos_bufferfub2.h, Logical/BufferedFub/BufferFub2_c-api_c-api/BufferFub2/exos_bufferfub2.c, Logical/BufferedFub/BufferFub2_c-api_c-api/BufferFub2/heapsize.cpp, Logical/BufferedFub/BufferFub2_c-api_c-api/Linux/termination.h, Logical/BufferedFub/BufferFub2_c-api_c-api/Linux/termination.c, Logical/BufferedFub/BufferFub_c-static_c-api/BufferFub/BufferFub.typ, Logical/BufferedFub/BufferFub_c-static_c-api/BufferFub/exos_bufferfub.c, Logical/BufferedFub/BufferFub_c-static_c-api/BufferFub/BufferFub.fun, Logical/BufferedFub/BufferFub_c-static_c-api/BufferFub/bufferfub.c, Logical/BufferedFub/BufferFub_c-static_c-api/BufferFub/heapsize.cpp, Logical/BufferedFub/BufferFub_c-static_c-api/BufferFub/libbufferfub.c, Logical/BufferedFub/BufferFub_c-static_c-api/BufferFub_0/BufferFub.st, Logical/BufferedFub/BufferFub_cpp_c-api/BufferFub_0, Logical/BufferedFub/BufferFub_cpp_c-api/BufferFub/BufferFub.typ, Logical/BufferedFub/BufferFub_cpp_c-api/BufferFub/exos_bufferfub.h, Logical/BufferedFub/BufferFub_cpp_c-api/BufferFub/BufferFub.fun, Logical/BufferedFub/BufferFub_cpp_c-api/BufferFub/bufferfub.cpp, Logical/BufferedFub/BufferFub_cpp_c-api/BufferFub/heapsize.cpp, Logical/BufferedFub/BufferFub_cpp_c-api/BufferFub/BufferFubDatamodel.hpp, Logical/BufferedFub/BufferFub_cpp_c-api/BufferFub/BufferFubDatamodel.cpp, Logical/BufferedFub/BufferFub_cpp_c-api/Linux/exos_bufferfub.h, Logical/BufferedFub/BufferFub_cpp_c-api/Linux/exos_bufferfub.c, Logical/BufferedFub/BufferFub_cpp_c-api/Linux/bufferfub.c, Logical/BufferedFub/BufferFub_cpp_c-api/Linux/termination.h, Logical/BufferedFub/BufferFub_cpp_c-api/Linux/termination.c, Logical/TemplateGen
